KUKA KRL program: ChillerOff.src

&ACCESS RVP
&REL 23
&PARAM EDITMASK = *
&PARAM TEMPLATE = C:\KRC\Roboter\Template\vorgabe
DEF ChillerOff( )

;************************************************
;              CNC Robotics Ltd
;              www.cncrobotics.co.uk
;************************************************
;     Contact: helpdesk@cncrobotics.co.uk
;     Date: 25/09/23
;     Version: 0.22.46
;************************************************
; Description: Routine to turn off the spindle
;************************************************
bRequestChiller =FALSE
WAIT FOR oCoolantOn==FALSE
bChillerRunning =FALSE
END
